FUNCTION WRITE_ANY_WORD : BOOL
VAR_INPUT
    ptr: POINTER TO WORD;
    val: WORD;
END_VAR

ptr^ := val;

END_FUNCTION

(* stored: Version 1.1.0.1, ProductVersion 3.1.4022.9
   POU WRITE_ANY_WORD: Id {00031d54-f0f1-405a-8c1e-ac2fc1af74f9}, SpecialFunc None *)
